// SIMATIC S7-200 project (STEP 7-Micro/WIN), CPU 224 REL 01.22

ORGANIZATION_BLOCK MAIN:OB1
TITLE=PROGRAM COMMENTS
BEGIN
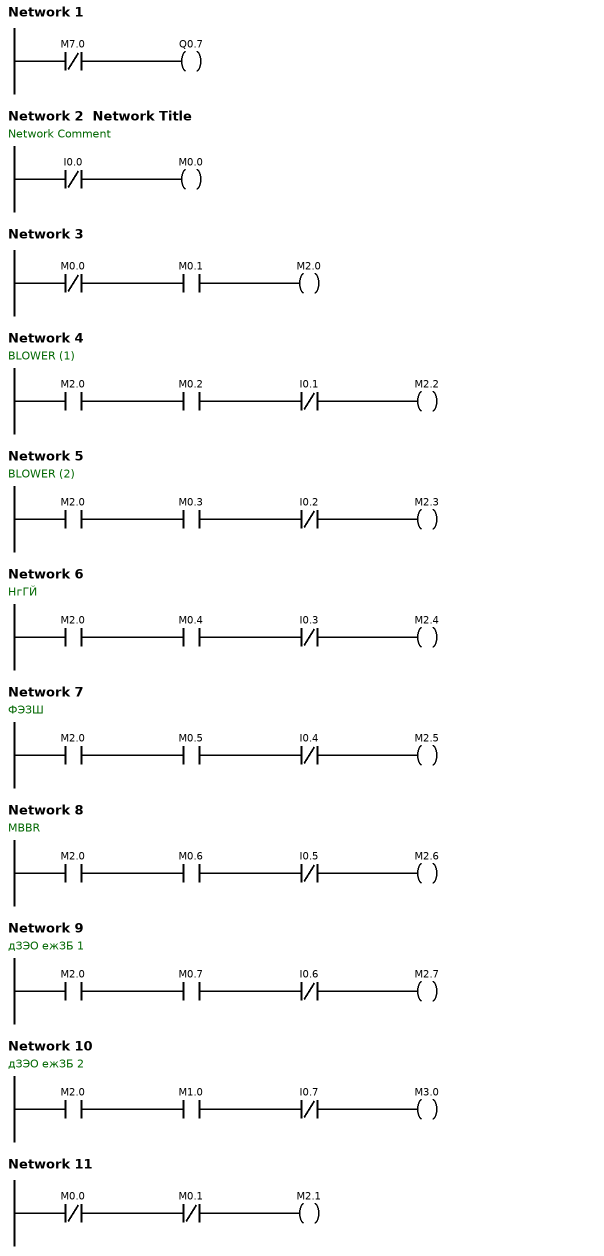
Network 1
LDN    M7.0
=      Q0.7
Network 2 // Network Title
// Network Comment
LDN    I0.0
=      M0.0
Network 3
LDN    M0.0
A      M0.1
=      M2.0
Network 4
// BLOWER (1)
LD     M2.0
A      M0.2
AN     I0.1
=      M2.2
Network 5
// BLOWER (2)
LD     M2.0
A      M0.3
AN     I0.2
=      M2.3
Network 6
// НгГЙ
LD     M2.0
A      M0.4
AN     I0.3
=      M2.4
Network 7
// ФЭЗШ
LD     M2.0
A      M0.5
AN     I0.4
=      M2.5
Network 8
// MBBR
LD     M2.0
A      M0.6
AN     I0.5
=      M2.6
Network 9
// дЗЭО ежЗБ 1
LD     M2.0
A      M0.7
AN     I0.6
=      M2.7
Network 10
// дЗЭО ежЗБ 2
LD     M2.0
A      M1.0
AN     I0.7
=      M3.0
Network 11
LDN    M0.0
AN     M0.1
=      M2.1
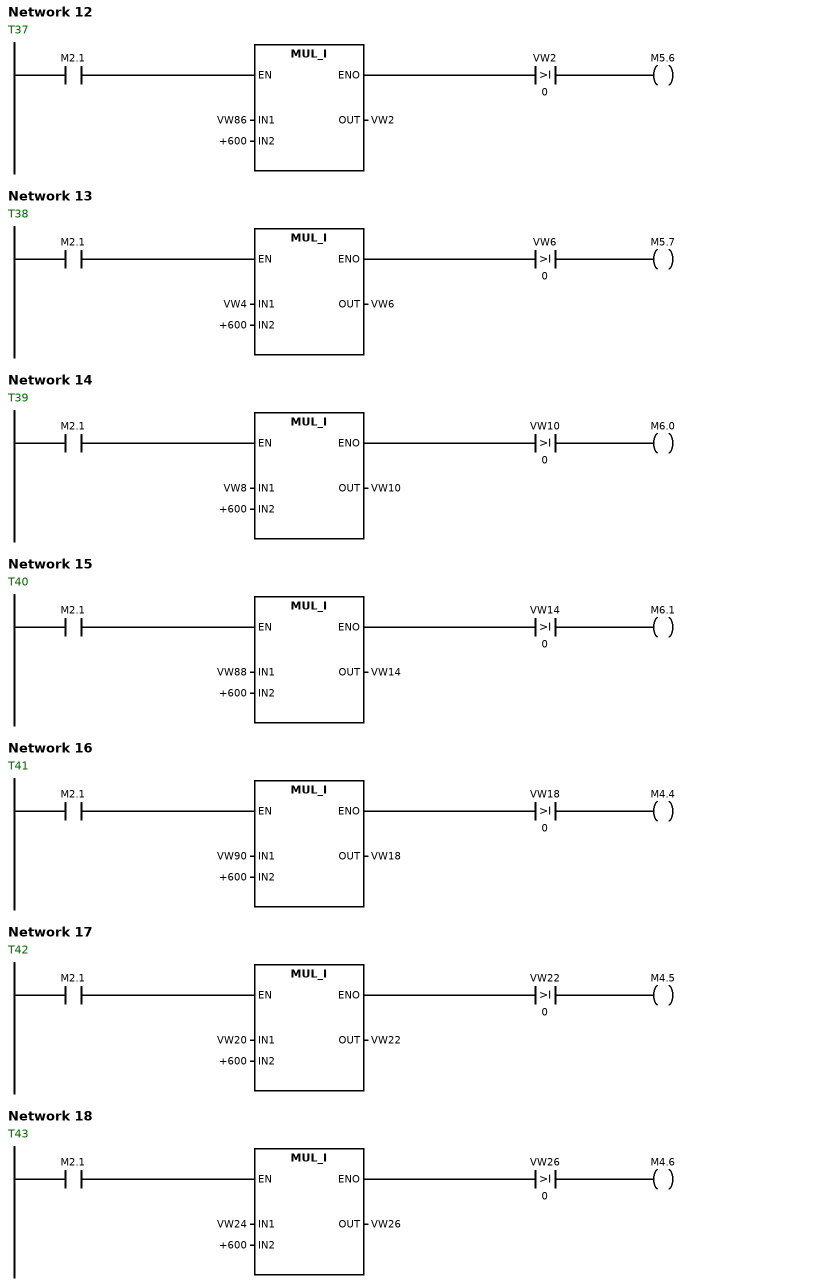
Network 12
// T37
LD     M2.1
MOVW   VW86, VW2
AENO
*I     +600, VW2
AENO
AW>    VW2, 0
=      M5.6
Network 13
// T38
LD     M2.1
MOVW   VW4, VW6
AENO
*I     +600, VW6
AENO
AW>    VW6, 0
=      M5.7
Network 14
// T39
LD     M2.1
MOVW   VW8, VW10
AENO
*I     +600, VW10
AENO
AW>    VW10, 0
=      M6.0
Network 15
// T40
LD     M2.1
MOVW   VW88, VW14
AENO
*I     +600, VW14
AENO
AW>    VW14, 0
=      M6.1
Network 16
// T41
LD     M2.1
MOVW   VW90, VW18
AENO
*I     +600, VW18
AENO
AW>    VW18, 0
=      M4.4
Network 17
// T42
LD     M2.1
MOVW   VW20, VW22
AENO
*I     +600, VW22
AENO
AW>    VW22, 0
=      M4.5
Network 18
// T43
LD     M2.1
MOVW   VW24, VW26
AENO
*I     +600, VW26
AENO
AW>    VW26, 0
=      M4.6
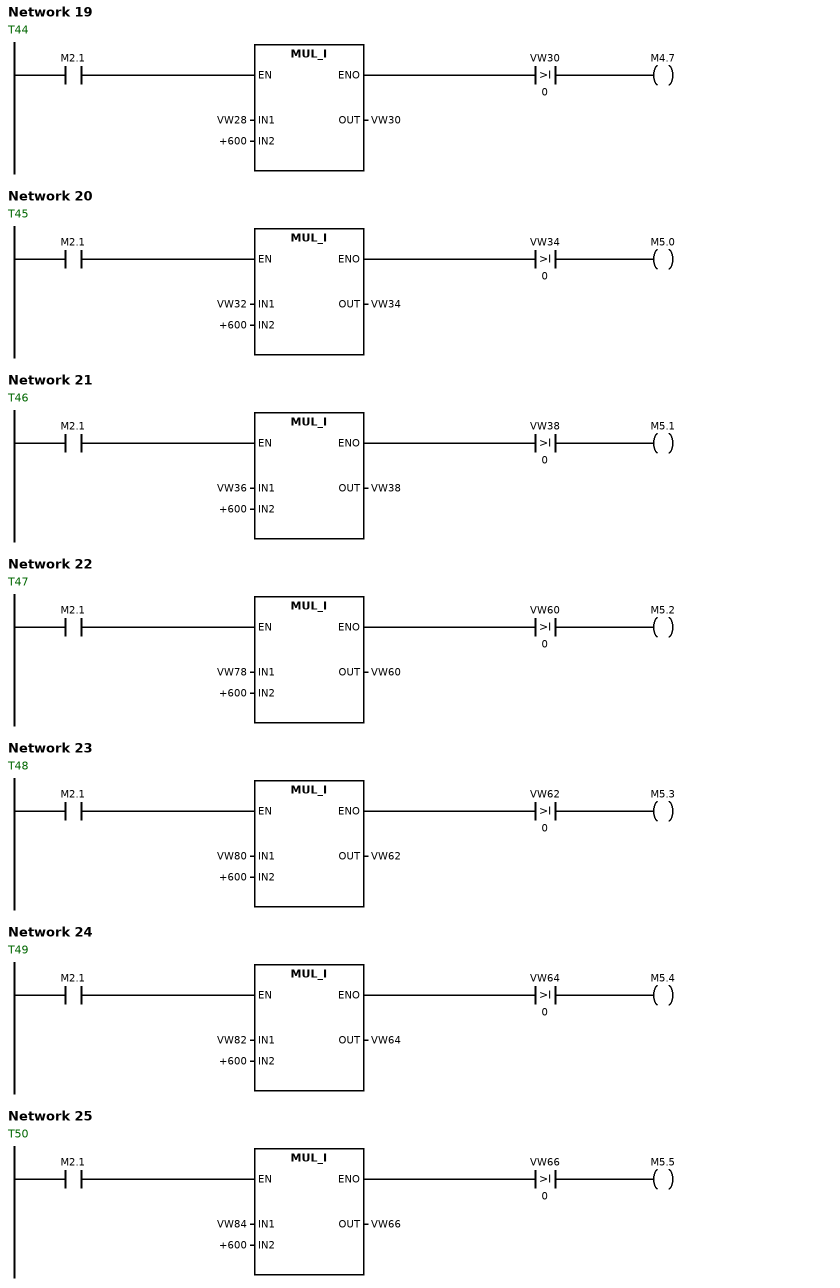
Network 19
// T44
LD     M2.1
MOVW   VW28, VW30
AENO
*I     +600, VW30
AENO
AW>    VW30, 0
=      M4.7
Network 20
// T45
LD     M2.1
MOVW   VW32, VW34
AENO
*I     +600, VW34
AENO
AW>    VW34, 0
=      M5.0
Network 21
// T46
LD     M2.1
MOVW   VW36, VW38
AENO
*I     +600, VW38
AENO
AW>    VW38, 0
=      M5.1
Network 22
// T47
LD     M2.1
MOVW   VW78, VW60
AENO
*I     +600, VW60
AENO
AW>    VW60, 0
=      M5.2
Network 23
// T48
LD     M2.1
MOVW   VW80, VW62
AENO
*I     +600, VW62
AENO
AW>    VW62, 0
=      M5.3
Network 24
// T49
LD     M2.1
MOVW   VW82, VW64
AENO
*I     +600, VW64
AENO
AW>    VW64, 0
=      M5.4
Network 25
// T50
LD     M2.1
MOVW   VW84, VW66
AENO
*I     +600, VW66
AENO
AW>    VW66, 0
=      M5.5
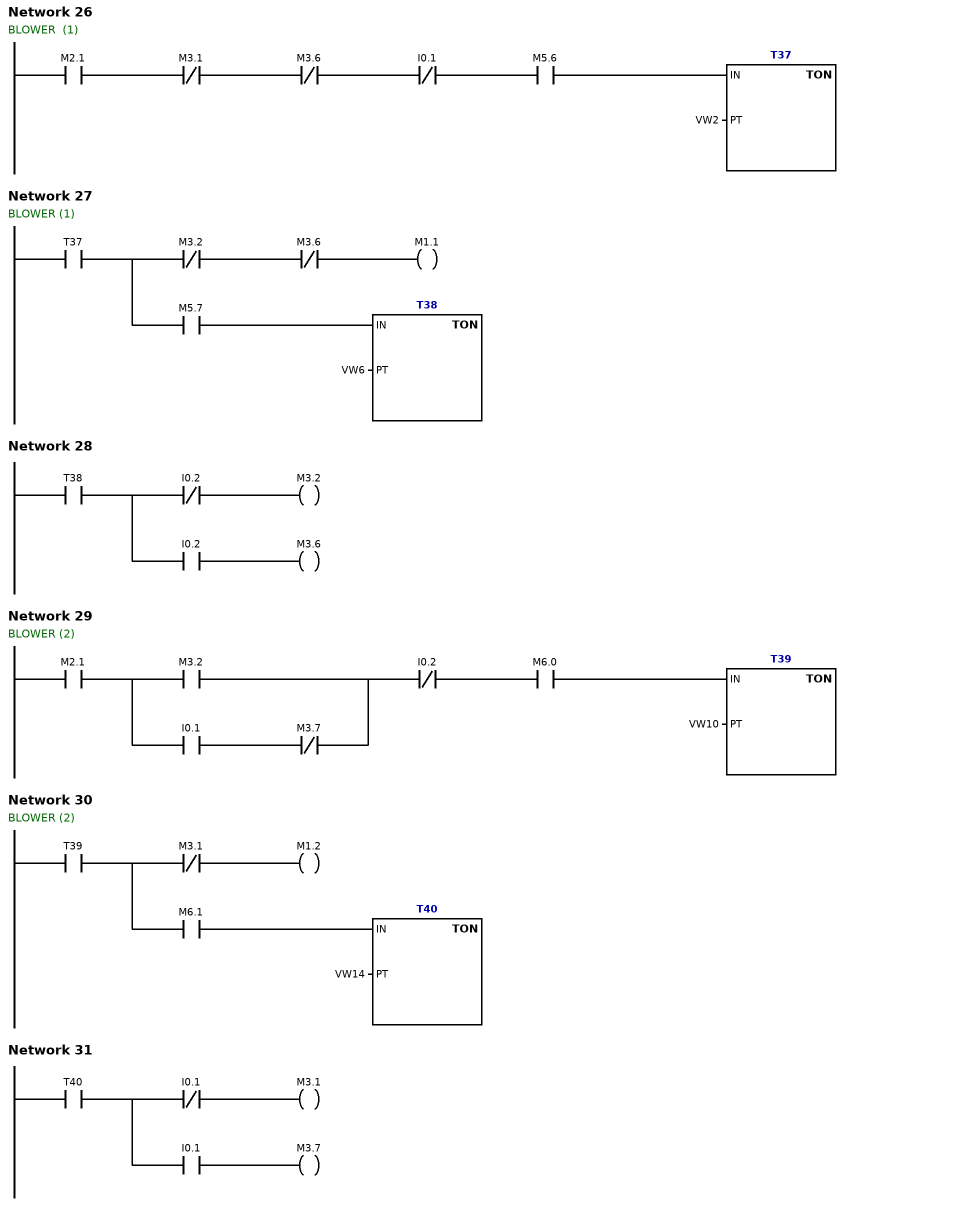
Network 26
// BLOWER  (1)
LD     M2.1
AN     M3.1
AN     M3.6
AN     I0.1
A      M5.6
TON    T37, VW2
Network 27
// BLOWER (1)
LD     T37
LPS
AN     M3.2
AN     M3.6
=      M1.1
LPP
A      M5.7
TON    T38, VW6
Network 28
LD     T38
LPS
AN     I0.2
=      M3.2
LPP
A      I0.2
=      M3.6
Network 29
// BLOWER (2)
LD     M2.1
LD     M3.2
LD     I0.1
AN     M3.7
OLD
ALD
AN     I0.2
A      M6.0
TON    T39, VW10
Network 30
// BLOWER (2)
LD     T39
LPS
AN     M3.1
=      M1.2
LPP
A      M6.1
TON    T40, VW14
Network 31
LD     T40
LPS
AN     I0.1
=      M3.1
LPP
A      I0.1
=      M3.7
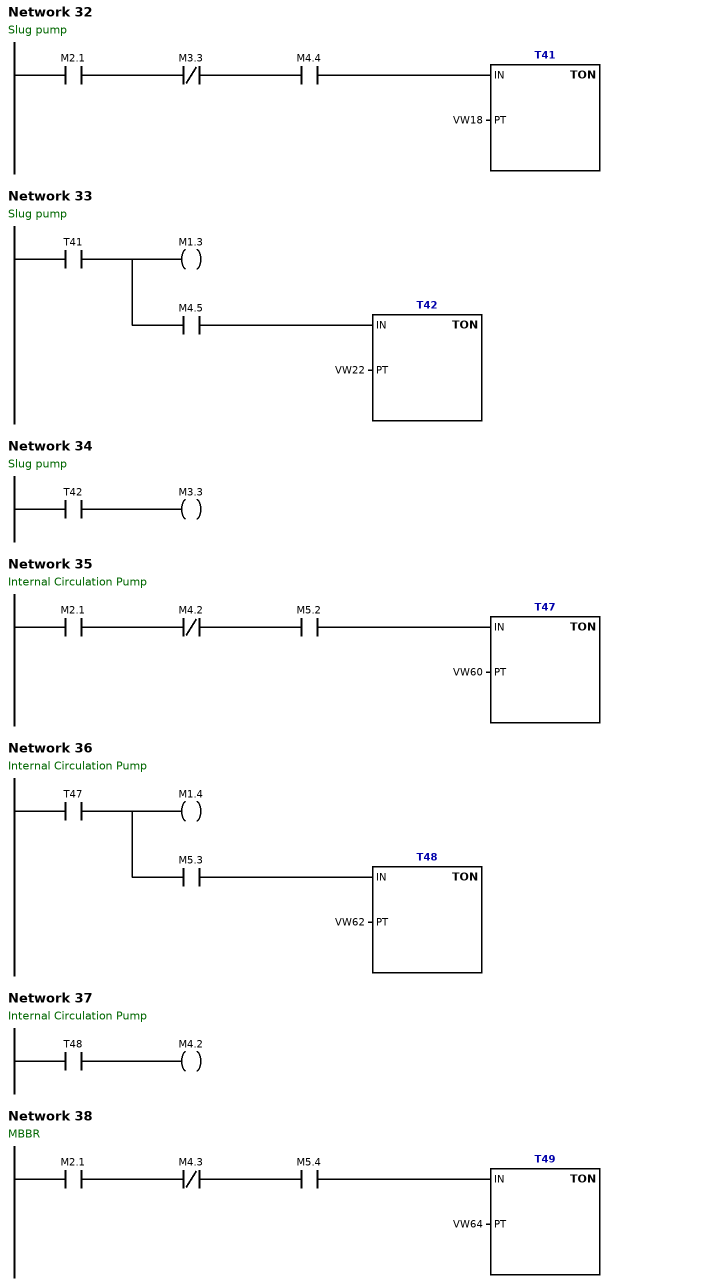
Network 32
// Slug pump
LD     M2.1
AN     M3.3
A      M4.4
TON    T41, VW18
Network 33
// Slug pump
LD     T41
=      M1.3
A      M4.5
TON    T42, VW22
Network 34
// Slug pump
LD     T42
=      M3.3
Network 35
// Internal Circulation Pump
LD     M2.1
AN     M4.2
A      M5.2
TON    T47, VW60
Network 36
// Internal Circulation Pump
LD     T47
=      M1.4
A      M5.3
TON    T48, VW62
Network 37
// Internal Circulation Pump
LD     T48
=      M4.2
Network 38
// MBBR
LD     M2.1
AN     M4.3
A      M5.4
TON    T49, VW64
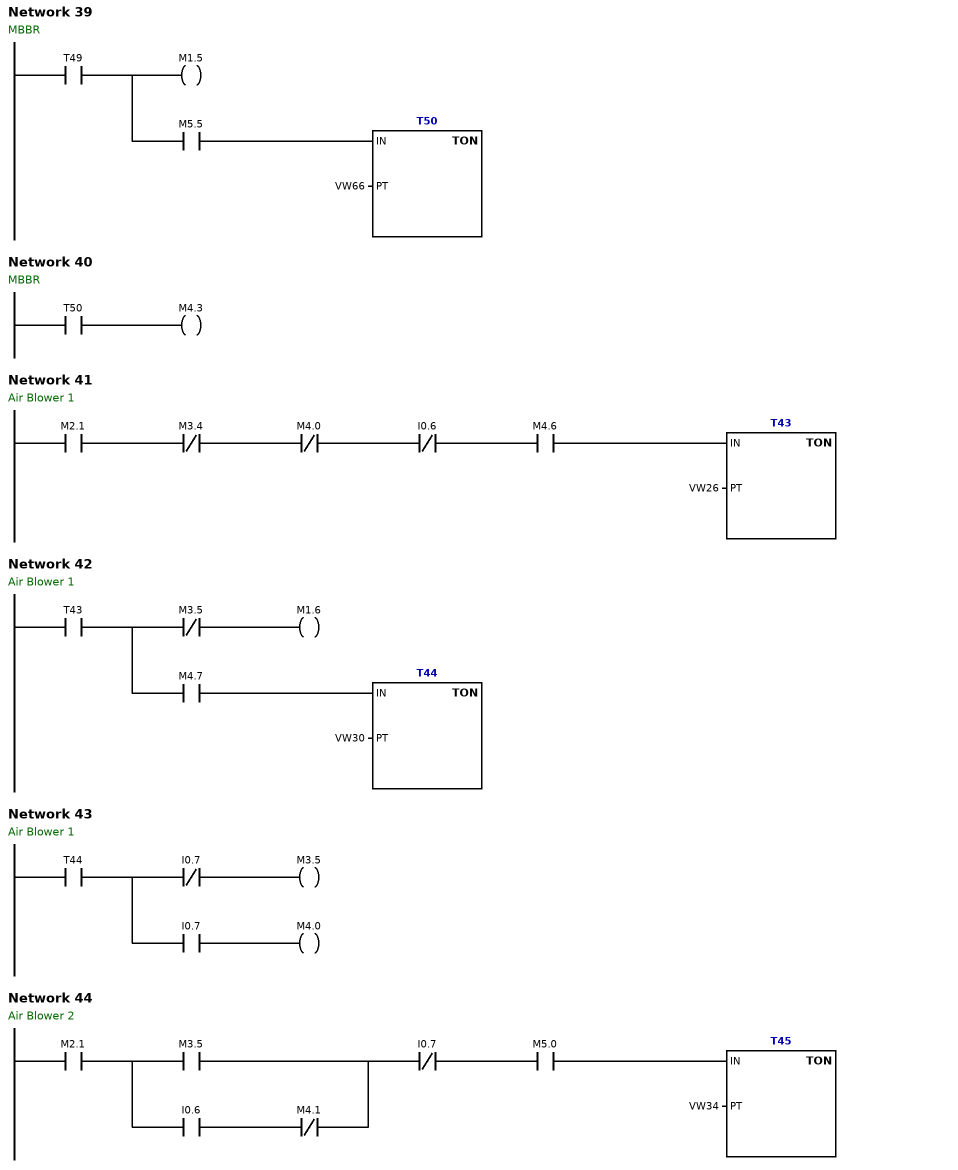
Network 39
// MBBR
LD     T49
=      M1.5
A      M5.5
TON    T50, VW66
Network 40
// MBBR
LD     T50
=      M4.3
Network 41
// Air Blower 1
LD     M2.1
AN     M3.4
AN     M4.0
AN     I0.6
A      M4.6
TON    T43, VW26
Network 42
// Air Blower 1
LD     T43
LPS
AN     M3.5
=      M1.6
LPP
A      M4.7
TON    T44, VW30
Network 43
// Air Blower 1
LD     T44
LPS
AN     I0.7
=      M3.5
LPP
A      I0.7
=      M4.0
Network 44
// Air Blower 2
LD     M2.1
LD     M3.5
LD     I0.6
AN     M4.1
OLD
ALD
AN     I0.7
A      M5.0
TON    T45, VW34
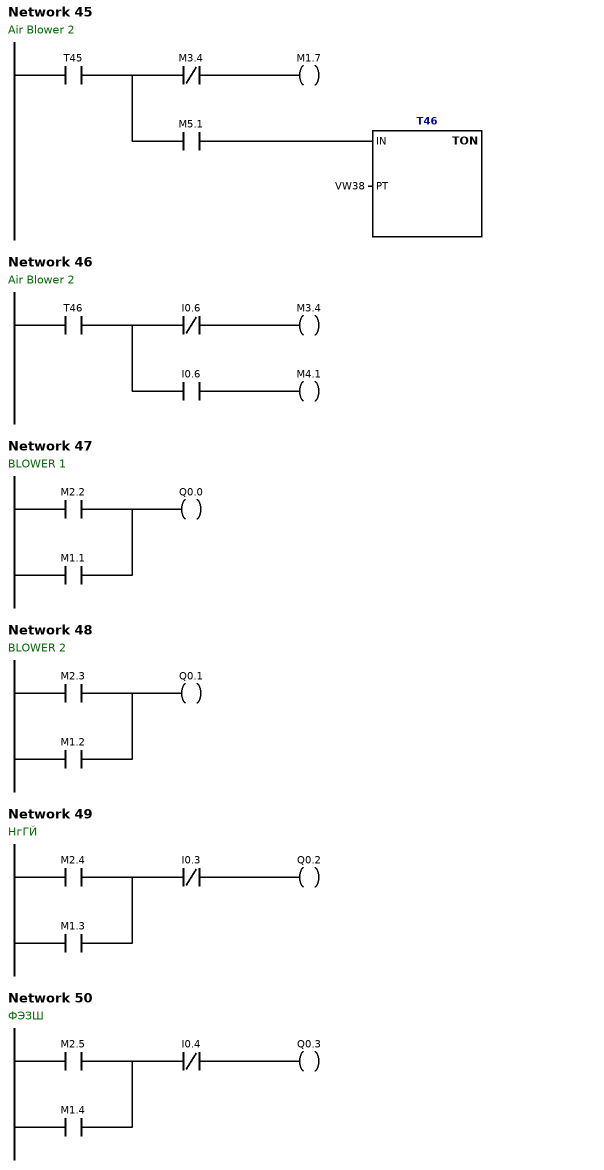
Network 45
// Air Blower 2
LD     T45
LPS
AN     M3.4
=      M1.7
LPP
A      M5.1
TON    T46, VW38
Network 46
// Air Blower 2
LD     T46
LPS
AN     I0.6
=      M3.4
LPP
A      I0.6
=      M4.1
Network 47
// BLOWER 1
LD     M2.2
O      M1.1
=      Q0.0
Network 48
// BLOWER 2
LD     M2.3
O      M1.2
=      Q0.1
Network 49
// НгГЙ
LD     M2.4
O      M1.3
AN     I0.3
=      Q0.2
Network 50
// ФЭЗШ
LD     M2.5
O      M1.4
AN     I0.4
=      Q0.3
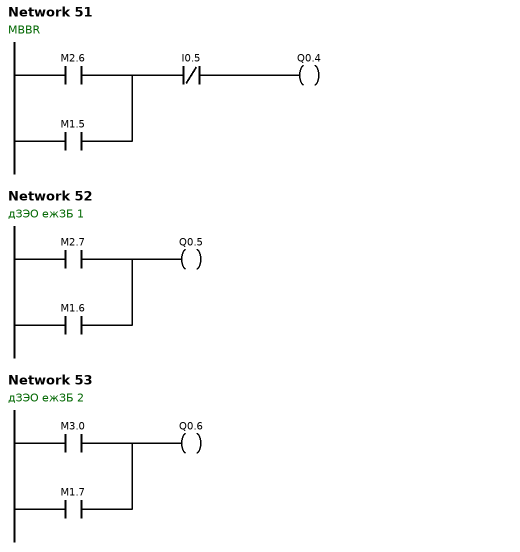
Network 51
// MBBR
LD     M2.6
O      M1.5
AN     I0.5
=      Q0.4
Network 52
// дЗЭО ежЗБ 1
LD     M2.7
O      M1.6
=      Q0.5
Network 53
// дЗЭО ежЗБ 2
LD     M3.0
O      M1.7
=      Q0.6
END_ORGANIZATION_BLOCK

SUBROUTINE_BLOCK SBR_0:SBR0
TITLE=SUBROUTINE COMMENTS
BEGIN
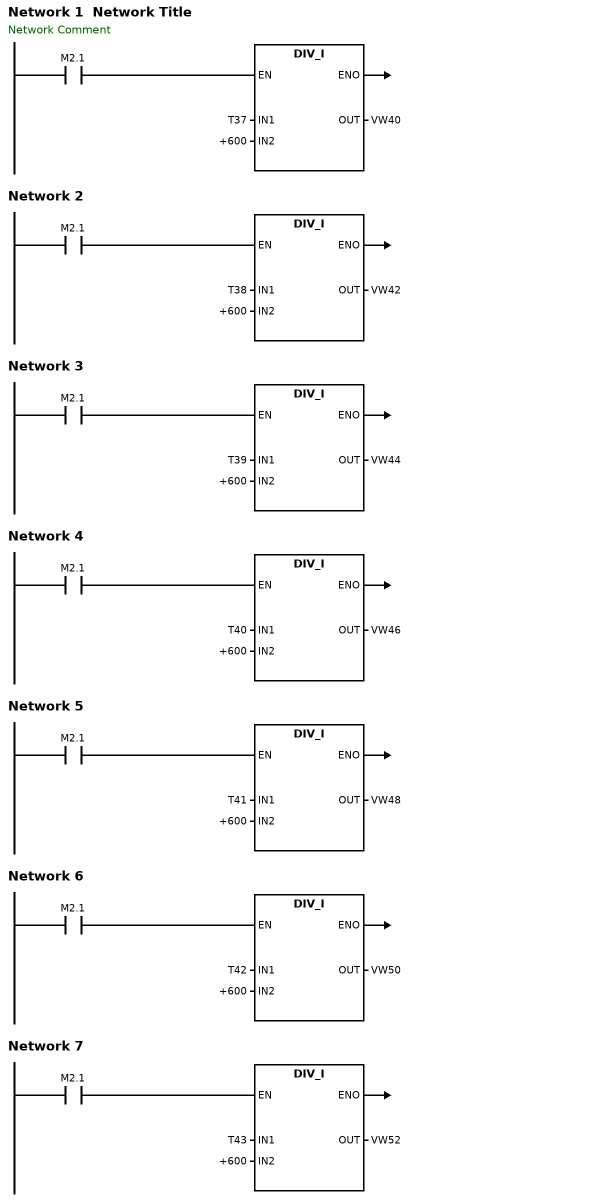
Network 1 // Network Title
// Network Comment
LD     M2.1
MOVW   T37, VW40
/I     +600, VW40
Network 2
LD     M2.1
MOVW   T38, VW42
/I     +600, VW42
Network 3
LD     M2.1
MOVW   T39, VW44
/I     +600, VW44
Network 4
LD     M2.1
MOVW   T40, VW46
/I     +600, VW46
Network 5
LD     M2.1
MOVW   T41, VW48
/I     +600, VW48
Network 6
LD     M2.1
MOVW   T42, VW50
/I     +600, VW50
Network 7
LD     M2.1
MOVW   T43, VW52
/I     +600, VW52
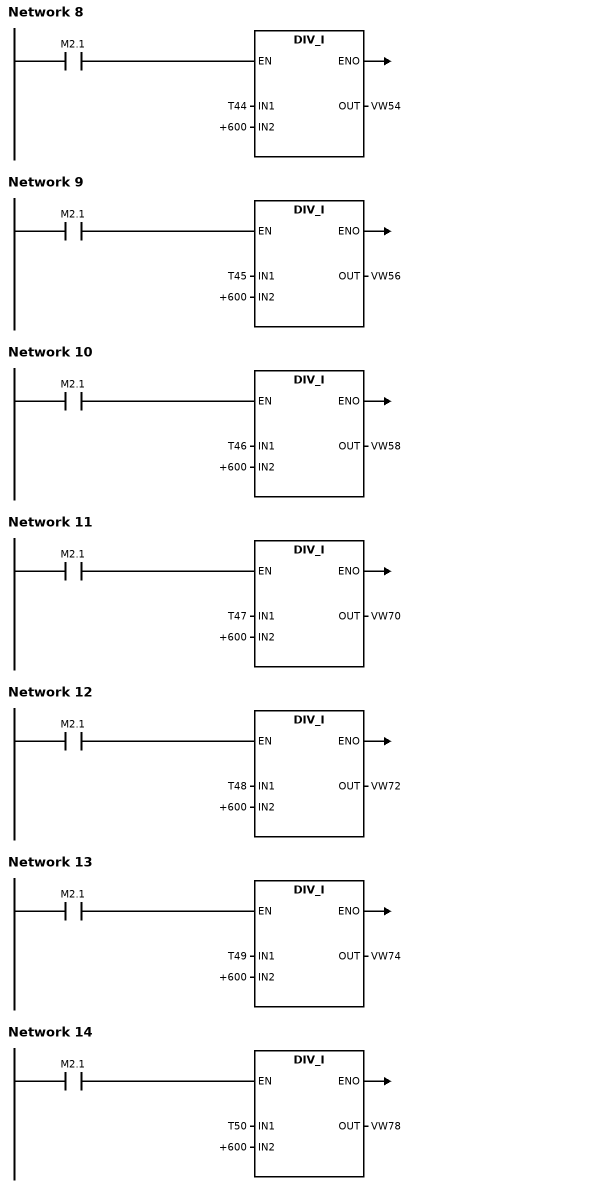
Network 8
LD     M2.1
MOVW   T44, VW54
/I     +600, VW54
Network 9
LD     M2.1
MOVW   T45, VW56
/I     +600, VW56
Network 10
LD     M2.1
MOVW   T46, VW58
/I     +600, VW58
Network 11
LD     M2.1
MOVW   T47, VW70
/I     +600, VW70
Network 12
LD     M2.1
MOVW   T48, VW72
/I     +600, VW72
Network 13
LD     M2.1
MOVW   T49, VW74
/I     +600, VW74
Network 14
LD     M2.1
MOVW   T50, VW78
/I     +600, VW78
END_SUBROUTINE_BLOCK
